{attribute addProperty BoxType "EL5152-0000-0018"}
{attribute addProperty Id "StatusAT %I*Status_FFD656FC1620Counter_valueAT %I*UINT16217"}
{attribute addProperty CRC "3805319245"}
{attribute addProperty SizeInBites "32"}
{attribute addProperty SizeInBytes "4"}
TYPE ENC_Status_compact_Channel_E2D0904D :
STRUCT
	{attribute addProperty Name "Status"}
	Status AT %I* : Status_FFD656FC;
	{attribute addProperty Name "Counter_value"}
	Counter_value AT %I* : UINT;
END_STRUCT
END_TYPE

(* stored: Version 1.2.0.0, ProductVersion 3.1.4024.9
   DUT ENC_Status_compact_Channel_E2D0904D: Id {47553334-f99a-4ef9-aa13-2bf311b2e37f} *)
